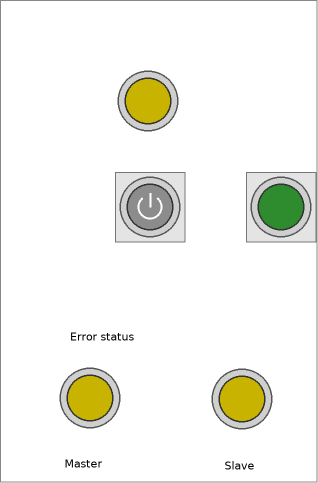
VISUALIZATION Visualization  // 318x483
    Lamp1 (113,66 70x70), variable: MAIN.fb_masterPower.Status, style: Lamp-Lamp1-Yellow
    PowerSwitch (115,172 70x70), variable: MAIN.bPower, behaviour: TOGGLE, style: Switch-PowerSwitch-Gray
    Lamp1 (55,363 70x70), variable: MAIN.fb_masterStatus.Error, style: Lamp-Lamp1-Yellow
    Lamp1 (207,364 70x70), variable: MAIN.fb_slaveStatus.Error, style: Lamp-Lamp1-Yellow
    Label (39,449 89x30), "Master"
    Label (197,451 85x30), "Slave"
    Label (54,322 96x30), "Error status"
    PushSwitch (246,172 70x70), variable: MAIN.bMove, behaviour: TAP, style: Switch-PushSwitch-Green
END_VISUALIZATION

(* stored: Version 1.1.0.1, ProductVersion 3.1.4022.17
   Visu Visualization: Id {9c176150-72ad-41ed-baed-7a970988747c} *)
